FUNCTION_BLOCK T_PMLSubUnitInfo IMPLEMENTS I_PMLSubUnitInfo
VAR
	_info : ST_PMLSubUnitInfo;
END_VAR

PROPERTY Info : REFERENCE TO ST_PMLSubUnitInfo
GET
Info REF= _info;
END_GET
END_PROPERTY

END_FUNCTION_BLOCK

(* stored: Version 1.1.0.1, ProductVersion 3.1.4024.12
   POU T_PMLSubUnitInfo: Id {f3d6df37-5abe-48ff-8f9b-c12aac828f4c}, SpecialFunc None
   Property Info: Id {f63d9b5b-4ac5-416f-8f67-e01104a54ab1}
   Get Get: Id {dc68f62b-a985-49b1-91f0-fe75bc53699c} *)
